
FUNCTION CB_byte_to_dword : DWORD

TITLE = ' Convert a byte into a Dword '
VERSION : '1.0'
AUTHOR  : CB
NAME    : bytToDwo
FAMILY  : TNI

VAR_INPUT
    IN : BYTE;
END_VAR

BEGIN

CB_byte_to_dword := BYTE_TO_DWORD(IN);

END_FUNCTION
